(* IEC 61131-3 sources: PLC_ST_Simulator/src/lib/library/standard, 15 files *)

(* ---- FbAxisAbs.st ---- *)
FUNCTION_BLOCK FbAxisAbs
    VAR_INPUT
        iAct : BOOL;
        iAxisNo : INT;
        iSpeed : INT;
        iStop : BOOL;
        iDest : DINT;
    END_VAR
    VAR_OUTPUT
        oBusy : BOOL;
        oDone : BOOL;
        oErr : BOOL;
    END_VAR
    VAR
        done : BOOL;
        (* Mock Logic *)
        tmrDelay : TON;
    END_VAR

    (* Mock Implementation *)
    IF iAct AND NOT oBusy AND NOT oDone THEN
        oBusy := TRUE;
        oErr := FALSE;
    END_IF;

    IF oBusy THEN
        tmrDelay(IN := TRUE, PT := T#500ms);
        IF tmrDelay.Q THEN
            oBusy := FALSE;
            oDone := TRUE;
            tmrDelay(IN := FALSE);
        END_IF;
    ELSE
        tmrDelay(IN := FALSE);
    END_IF;

    IF NOT iAct THEN
        oDone := FALSE;
    END_IF;
END_FUNCTION_BLOCK

(* ---- FbAxisZero.st ---- *)
FUNCTION_BLOCK FbAxisZero
    VAR_INPUT
        iAct : BOOL;
        iAxisNo : INT; (* WORD/Bit String 16 *)
        iHomeSpeed : INT;
        iApproachSpeed : INT;
        iStop : BOOL;
    END_VAR
    VAR_OUTPUT
        oBusy : BOOL;
        oDone : BOOL;
        oErr : BOOL;
    END_VAR
    VAR
        done : BOOL;
        (* Mock Logic *)
        step : INT := 0;
        tmrDelay : TON;
    END_VAR

    (* Mock Implementation *)
    IF iAct AND NOT oBusy AND NOT oDone THEN
        oBusy := TRUE;
        oErr := FALSE;
        step := 1;
    END_IF;

    IF oBusy THEN
        tmrDelay(IN := TRUE, PT := T#1s);
        IF tmrDelay.Q THEN
            oBusy := FALSE;
            oDone := TRUE;
            tmrDelay(IN := FALSE);
        END_IF;
    ELSE
        tmrDelay(IN := FALSE);
    END_IF;

    IF NOT iAct THEN
        oDone := FALSE;
    END_IF;

END_FUNCTION_BLOCK

(* ---- FbCylinder0x1y.st ---- *)
FUNCTION_BLOCK FbCylinder0x1y
    VAR_INPUT
        iAct : BOOL; (* Action Cmd *)
        iOnDelay : INT; (* Sensor On Delay *)
        iOffDelay : INT; (* Sensor Off Delay *)
    END_VAR
    VAR_OUTPUT
        oDevice : BOOL; (* Target Device *)
        oOn : BOOL;
        oOff : BOOL;
    END_VAR
    VAR
        tmrOnDelay : TON;
        tmrOffDelay : TON;
    END_VAR

    oDevice := iAct;

    tmrOnDelay(IN := oDevice, PT := INT_TO_TIME(iOnDelay*10));
    oOn := tmrOnDelay.Q;

    tmrOffDelay(IN := NOT oDevice, PT := INT_TO_TIME(iOffDelay*10));
    oOff := tmrOffDelay.Q;

END_FUNCTION_BLOCK

(* ---- FbCylinder1x1y.st ---- *)
FUNCTION_BLOCK FbCylinder1x1y
    VAR_INPUT
        iAct : BOOL;
        iRst : BOOL;
        iOnDelay : INT;
        iOffDelay : INT;
        iOnTO : INT;
        iOffTO : INT;
        iLimit1 : BOOL;
    END_VAR
    VAR_OUTPUT
        oDevice : BOOL;
        oOn : BOOL;
        oOff : BOOL;
        oErr : BOOL;
        oErrId : INT;
    END_VAR
    VAR
        tmrOn : TON;
        tmrOff : TON;
        tmrOnDelay : TON;
        tmrOffDelay : TON;
    END_VAR

    oDevice := iAct;

    tmrOn(IN := oDevice AND NOT iLimit1, PT:= INT_TO_TIME(iOnTO*10));
    tmrOff(IN := NOT oDevice AND iLimit1, PT:= INT_TO_TIME(iOffTO*10));

    IF iRst AND oErr THEN
        oErr := FALSE;
    END_IF;

    IF tmrOn.Q OR tmrOff.Q THEN
        oErr := TRUE;
    END_IF;

    IF oErr THEN
        IF tmrOff.Q THEN
            oErrId := 20;
        ELSIF tmrOn.Q THEN
            oErrId := 10;
        END_IF;
    ELSE
        oErrId := 0;
    END_IF;

    tmrOnDelay(IN := oDevice AND iLimit1, PT := INT_TO_TIME(iOnDelay*10));
    oOn := tmrOnDelay.Q;

    tmrOffDelay(IN := NOT oDevice, PT := INT_TO_TIME(iOffDelay*10));
    oOff := tmrOffDelay.Q;

END_FUNCTION_BLOCK

(* ---- FbCylinder2x1y.st ---- *)
FUNCTION_BLOCK FbCylinder2x1y
    VAR_INPUT
        iAct : BOOL;
        iRst : BOOL;
        iOnDelay : INT;
        iOffDelay : INT;
        iOnTO : INT;
        iOffTO : INT;
        iLimit1 : BOOL;
        iLimit2 : BOOL;
    END_VAR
    VAR_OUTPUT
        oDevice : BOOL;
        oOn : BOOL;
        oOff : BOOL;
        oErr : BOOL;
        oErrId : INT;
    END_VAR
    VAR
        tmrOn : TON;
        tmrOff : TON;
        tmrErr : TON;
        tmrOnDelay : TON;
        tmrOffDelay : TON;
    END_VAR

    oDevice := iAct;

    tmrOn(IN := oDevice AND NOT iLimit2, PT:= INT_TO_TIME(iOnTO * 10));
    tmrOff(IN := NOT oDevice AND NOT iLimit1, PT := INT_TO_TIME(iOffTO * 10));
    tmrErr(IN := iLimit1 AND iLimit2, PT := T#10s);

    IF iRst AND oErr THEN
        oErr := FALSE;
    END_IF;

    IF tmrOn.Q OR tmrOff.Q OR tmrErr.Q THEN
        oErr := TRUE;
    END_IF;

    IF (oErr) THEN
        IF tmrOn.Q THEN
            oErrId := 10;
        ELSIF  tmrOff.Q THEN
            oErrId := 20;
        END_IF;

        IF tmrErr.Q THEN
            oErrId := 30;
        END_IF;
    ELSE
        oErrId := 0;
    END_IF;

    tmrOnDelay(IN := oDevice AND iLimit2, PT := INT_TO_TIME(iOnDelay*10));
    oOn := tmrOnDelay.Q;

    tmrOffDelay(IN := NOT oDevice AND iLimit1, PT := INT_TO_TIME(iOffDelay*10));
    oOff := tmrOffDelay.Q;

END_FUNCTION_BLOCK

(* ---- FbFeeder.st ---- *)
FUNCTION_BLOCK FbFeeder
    VAR_INPUT
        iAct : BOOL;
        iFull : BOOL;
        iArrived : BOOL;
        iFullOnT : INT;
        iFullOffT : INT;
        iArrivedOnT : INT;
        iSupplyTO : INT;
        iArriveTO : INT;
    END_VAR
    VAR_OUTPUT
        oFeeder : BOOL;
        oLinearFeeder : BOOL;
        oCanPick : BOOL;
        oNeedSupply : BOOL;
        oArriveTO : BOOL;
    END_VAR
    VAR
        tmrArrivedOn : TON;
        tmrFullOn : TON;
        tmrNeedSupply : TON;
        tmrFullOff : TON;
        tmrArriveTO : TON;

        (* Edge helpers *)
        trigFullOff : R_TRIG;
        trigFullOn : R_TRIG;
    END_VAR

    oLinearFeeder := iAct;

    tmrArriveTO(
        IN := iAct AND NOT iArrived,
        PT := INT_TO_TIME(iArriveTO*100));

    tmrArrivedOn(
        IN := iAct AND iArrived,
        PT := INT_TO_TIME(iArrivedOnT*100));

    oCanPick := iAct AND tmrArrivedOn.Q;

    tmrFullOn(
        IN := iAct AND iFull,
        PT := INT_TO_TIME(iFullOnT*100));

    tmrFullOff(
        IN := iAct AND NOT iFull,
        PT := INT_TO_TIME(iFullOffT*100));

    (* Calculate edges *)
    trigFullOff(CLK := tmrFullOff.Q);
    trigFullOn(CLK := tmrFullOn.Q);

    IF iAct THEN
        IF trigFullOff.Q THEN
            oFeeder := TRUE; (* SET *)
        END_IF;

        IF trigFullOn.Q THEN
            oFeeder := FALSE; (* RST *)
        END_IF;
    ELSE
        oFeeder := FALSE; (* RST *)
    END_IF;

    tmrNeedSupply(
        IN := iAct AND oFeeder,
        PT := INT_TO_TIME(iSupplyTO*100));

    oNeedSupply := iAct AND tmrNeedSupply.Q AND (NOT tmrFullOn.Q);

    oArriveTO := tmrArriveTO.Q;

END_FUNCTION_BLOCK

(* ---- FbRotateTable.st ---- *)
FUNCTION_BLOCK FbRotateTable
    VAR_INPUT
        iOrigPos : BOOL;
        iActPos : BOOL;
        iStop : BOOL;
        iRun : BOOL;
        iReset : BOOL;
        iRotateTO : INT;
        iInPosWaitTime : INT;
    END_VAR
    VAR_OUTPUT
        oDevice : BOOL;
        oBusy : BOOL;
        oErr : BOOL;
        oArrived : BOOL;
    END_VAR
    VAR
        rotating : BOOL;
        tmrWaitInPos : TON;
        inPos : BOOL;
        waitInPos : BOOL;
        arrived : BOOL;
        rotate : BOOL;
        reset : BOOL;
        tmrTimeOut : TON;
        tmp : BOOL;

        (* Edge detection helpers *)
        trigRun : R_TRIG;
        trigOrigPos : R_TRIG;
    END_VAR

    (* Pre-calculate edges *)
    trigRun(CLK := iRun);
    rotate := trigRun.Q;
    trigOrigPos(CLK := iOrigPos);

    tmp := (NOT arrived) AND (NOT iStop) AND (rotate OR rotating);
    rotating := tmp;

    (* oDevice output calculation *)
    IF (NOT oErr) AND tmp THEN
        oDevice := TRUE;
    ELSE
        oDevice := FALSE;
    END_IF;

    reset := iReset;
    tmrTimeOut(IN := oDevice AND NOT reset, PT := INT_TO_TIME(iRotateTO * 100)); // Sample says *100? Assuming ms base

    IF NOT reset AND (tmrTimeOut.Q OR oErr) THEN
        oErr := TRUE;
    ELSE
        (* Manual Reset logic might be needed if strictly following Latching logic,
           but here oErr := ... is assignment.
           Sample has oErr := ... (OR oErr), which is self-holding.
           In ST assignment: oErr := ... OR oErr works as hold. *)
         oErr := NOT reset AND (tmrTimeOut.Q OR oErr);
    END_IF;

    inPos := (NOT tmrWaitInPos.Q AND NOT iStop) OR ((rotating AND trigOrigPos.Q) OR inPos);

    waitInPos := (NOT tmrWaitInPos.Q) AND (((NOT iStop) OR ((rotating AND trigOrigPos.Q) OR inPos)) OR waitInPos);

    tmrWaitInPos(IN:= ((inPos AND waitInPos) OR arrived) AND NOT iStop AND NOT tmrWaitInPos.Q, PT := INT_TO_TIME(iInPosWaittime));

    arrived := ((inPos AND waitInPos) OR arrived) AND NOT iStop AND NOT tmrWaitInPos.Q;

    oBusy := rotating AND NOT arrived;

    (* SET/RST translations *)
    IF tmrWaitInPos.Q THEN
        oArrived := TRUE;
    END_IF;

    IF trigRun.Q THEN
        oArrived := FALSE;
    END_IF;

END_FUNCTION_BLOCK

(* ---- FbSysStateProcess.st ---- *)
FUNCTION_BLOCK FbSysStateProcess
    VAR_IN_OUT
        // iStatus : dsSysStatus;
        // iTrig : dsSysTrigger;
    END_VAR

    (* Mock logic *)

END_FUNCTION_BLOCK

(* ---- FbTowerLight.st ---- *)
FUNCTION_BLOCK FbTowerLight
    VAR_INPUT
        // iStatus : dsSysStatus; (* STRUCT not fully supported in simple string parse unless defined *)
        iStopBuzzer : BOOL;
    END_VAR
    VAR_OUTPUT
        // oLights : dsTowerLight;
        hasErr : BOOL;
    END_VAR
    VAR
        keepStopBuzzer : BOOL;
    END_VAR

    (* Mock logic since structs are tricky in this simple setup *)
    hasErr := FALSE;

END_FUNCTION_BLOCK

(* ---- Always.st ---- *)
VAR
    calcA1Speed : BOOL;
    calcA2Speed : BOOL;
    a2HadDone : BOOL;
    axis2ZeroIdx : INT;
    axis1ZeroIdx : INT;
    tmpBool : BOOL;
    st3NextPosIdx : INT;
    manSt5PF : BOOL;
    manSt5LF : BOOL;
    st3StepGoPosIdx : INT;
    idx : INT;
    tmrWaitLetAxis2Down : TON;

    (* Helper vars for edge detection *)
    trigManMode : R_TRIG;
    trigAutoMode : R_TRIG;
    trigSt10Chk : R_TRIG;
    trigFeeder : R_TRIG;
    trigFeederOff : R_TRIG;
    trigRun : R_TRIG;
    trigRotateArrived : R_TRIG;
END_VAR

    tmrSysInit(IN := SM8000, PT:= T#10s);

    sys.EMG := NOT xEmg OR F0;

    IF NOT tmrSysInit.Q THEN
        RETURN;
    END_IF;

    IF sys.EMG THEN
        gSt3NextSide := 0;
        gSt3NeedCheck := TRUE;
    END_IF;

    trigManMode(CLK := sys.ManMode);
    IF trigManMode.Q THEN
        St1PutDone := FALSE;
        St3Done := FALSE;
        St5PutDone := FALSE;
        St6Done := FALSE;
        St7Done := FALSE;
        St8GetDone := FALSE;
        St8NeedGet := FALSE;

        gSt1Seperate := FALSE;
        gSt5Seperate := FALSE;

        St8GetDone := FALSE;
    END_IF;

    (* ALTP(uiLight, yLight); *)
    (* Implementing ALTP (Alternate) logic manually or assuming ALTP FB exists,
       but standard ST doesn't have ALTP. Usage: Toggle yLight on rising edge of uiLight? *)
     (* Assuming uiLight is a button. We need a trigger. *)
     (* For simplicity, skipping ALTP or assuming native support if valid.
        Re-implementing as simple toggle for now: *)
     (* IF trigUiLight.Q THEN yLight := NOT yLight; END_IF; *)

    gAutoCanGoNext := NOT sys.HasError;

    gCanChangePage := gAllStCanCycle;

    tmrSt10Chk(IN:=xSt10Check AND gRotateArrived, PT:=T#0.5s);
    IF gRotateArrived THEN
        IF tmrSt10Chk.Q THEN
            F3 := TRUE;
        END_IF;
    END_IF;

    IF ((uiStartAuto AND (NOT sys.AutoMode)) OR gClearTool) AND
        NOT F3 THEN

        IF NOT sys.HasError AND
            NOT gWaitStopAuto AND gAllStCanCycle AND
            NOT F6 AND
            NOT F7 THEN
            sys.AutoMode := TRUE;
            sys.ManMode := FALSE;
        END_IF;
    END_IF;

    (* SET/RST logic conversion *)
    IF sys.AutoMode AND uiStopAuto AND NOT gWaitStopAuto THEN
        gWaitStopAuto := TRUE;
    END_IF;

    IF sys.AutoMode AND uiStopAuto AND gClearTool THEN
        gClearTool := FALSE;
    END_IF;

    IF uiClearTool AND NOT F3 THEN
        (* CheckHasTool is likely a function call *)
        (* IF CheckHasTool(wDataArray) THEN *)
        (* Assuming CheckHasTool returns BOOL *)
            gClearTool := TRUE;
        (* END_IF; *)
    END_IF;

    gAllStCycleDone :=
        (NOT St1Cycle OR St1PutDone) AND
        (NOT St3Cycle (* OR St3Done*)) AND
        (NOT St5Cycle OR St5PutDone) AND

        ((NOT UseSt6) OR
        (UseSt6 AND NOT St6Cycle)) AND

        NOT St7Cycle AND
        (NOT St8NeedGet OR (St8NeedGet AND St8GetDone)) AND
        NOT St9Cycle;

    gAllStCanCycle :=
        St1InOrg AND
        St3InOrg AND
        St5InOrg AND

        ((NOT UseSt6) OR
        (UseSt6 AND St6InOrg)) AND

        (* St7InOrg AND *)
        St8InOrg AND
        St9InOrg;

    gLight.Yellow :=
        F54 OR
        F55 OR
        F56 OR
        F57;

    gLight.Green :=
        (sys.ManMode AND SM8013) OR
        (sys.AutoMode);

    gLight.Red :=
        SM8013 AND (sys.EMG OR sys.HasError OR sys.HasWarning);

    gBuzzerEnable := NOT uiEnBuzzer;
    gLight.Buzzer := gBuzzerEnable AND
        SM8013 AND (sys.HasWarning OR sys.HasError);

    IF manRotate THEN
        gRotate := TRUE;
        manRotate := FALSE;
    END_IF;

    trigFeeder(CLK := uiFeeder);
    IF trigFeeder.Q THEN
        gSt1RotatoryFeeder := TRUE;
        gSt5RotatoryFeeder := TRUE;

        gSt3Feed := gAllAxisZeroDone AND gA1IO.xReady;
    END_IF;

    trigFeederOff(CLK := uiFeeder); (* This needs falling edge detection *)
    (* Actually LDF is Falling Edge. R_TRIG detects Rising.
       Need F_TRIG for LDF. *)
    (* F_TRIG declaration missing, using logic: *)
    IF (NOT uiFeeder) AND tmpBool(*prev*) THEN
        gSt1RotatoryFeeder := FALSE;
        gSt5RotatoryFeeder := FALSE;
        gSt3Feed := FALSE;

        gSt1Vacuum := FALSE;
        gSt5SquareVacuum := FALSE;
    END_IF;
    tmpBool := uiFeeder; (* Store for falling edge check next cycle *)

    IF gClearDataArray THEN
        FOR idx := 0 TO 9 BY 1 DO
            wDataArray[idx] := 0;
        END_FOR;
        gClearDataArray := FALSE;
    END_IF;

    RotateTable(
        iOrigPos:= xIndexOrg,
        iActPos:= xIndexAct,
        iRun:= gRotate AND (NOT sys.Error),
        iRotateTO:= wRotateTO,
        iInPosWaitTime:= wRotateOnPosWaitT,
        iReset := ResetAlarm,
        oDevice => yIndex);

    IF RotateTable.oBusy THEN
        gRotate := FALSE;
    END_IF;

    trigRotateArrived(CLK := RotateTable.oArrived);
    IF trigRotateArrived.Q THEN
        gRotateArrived := TRUE;
    END_IF;

    (* Cylinders *)
    cySt1Down(
        iAct := gSt1Down,
        iRst := ResetAlarm,
        iLimit1 := xSt1DownOrg,
        iLimit2 := xSt1DownAct,
        oDevice =>ySt1Down,
        iOnTO := wSt1DownTO,
        iOffTO := wSt1DownTO,
        iOnDelay := wSt1DownOnT,
        iOffDelay := wSt1DownOffT);

    cySt1Forward(
        iAct := gSt1Forward,
        iRst := ResetAlarm,
        iLimit1 := xSt1ForwardOrg,
        iLimit2 := xSt1ForwardAct,
        oDevice =>ySt1Forward,
        iOnTO := wSt1ForwardTO,
        iOffTO := wSt1ForwardTO,
        iOnDelay := wSt1ForwardOnT,
        iOffDelay := wSt1ForwardOffT);

    cySt1Clamp(
        iAct := gSt1Clamp,
        oDevice =>ySt1Clamp,
        iOnDelay := wSt1ClampOnT,
        iOffDelay := wSt1ClampOffT);

    cySt1ClampRotate(
        iAct := gSt1ClampRotate,
        iRst := ResetAlarm,
        iLimit1 := xSt1ClampRotateOrg,
        iLimit2 := xSt1ClampRotateAct,
        oDevice =>ySt1ClampRotate,
        iOnTO := wSt1ClampRotateTO,
        iOffTO := wSt1ClampRotateTO,
        iOnDelay := wSt1ClampRotateOnT,
        iOffDelay := wSt1ClampRotateOffT);

    cySt1Seperate(
        iAct := gSt1Seperate,
        iRst := ResetAlarm,
        iLimit1 := xSt1SeperateOrg,
        iLimit2 := xSt1SeperateAct,
        oDevice =>ySt1Seperate,
        iOnTO := wSt1SeperateTO,
        iOffTO := wSt1SeperateTO,
        iOnDelay := wSt1SeperateOnT,
        iOffDelay := wSt1SeperateOffT);

    cySt3Down(
        iAct := gSt3Down,
        iRst := ResetAlarm,
        iLimit1 := xSt3DownOrg,
        iLimit2 := xSt3DownAct,
        oDevice =>ySt3Down,
        iOnTO := wSt3DownTO,
        iOffTO := wSt3DownTO,
        iOnDelay := wSt3DownOnT,
        iOffDelay := wSt3DownOffT);

    cySt3Forward(
        iAct := gSt3Forward,
        iRst := ResetAlarm,
        iLimit1 := xSt3ForwardOrg,
        iLimit2 := xSt3ForwardAct,
        oDevice =>ySt3Forward,
        iOnTO := wSt3ForwardTO,
        iOffTO := wSt3ForwardTO,
        iOnDelay := wSt3ForwardOnT,
        iOffDelay := wSt3ForwardOffT);

    cySt3Suck(
        iAct := gSt3Suck,
        iRst := ResetAlarm,
        iLimit1 := xSt3SuckOrg,
        oDevice => ySt3Suck,
        iOnDelay := wSt3SuckOnT,
        iOffDelay := wSt3SuckOffT,
        iOnTO := wSt3SuckTO,
        iOffTO := wSt3SuckTO);

    cySt5Suck(
        iAct := gSt5Suck,
        iRst := ResetAlarm,
        iLimit1 := xSt5SuckOrg,
        oDevice => ySt5Vacuum,
        iOnDelay := wSt5SuckOnT,
        iOffDelay := wSt5SuckOffT,
        iOnTO := wSt5SuckTO,
        iOffTO := wSt5SuckTO);

    cySt5Down(
        iAct := gSt5Down,
        iRst := ResetAlarm,
        iLimit1 := xSt5DownOrg,
        iLimit2 := xSt5DownAct,
        oDevice =>ySt5Down,
        iOnTO := wSt5DownTO,
        iOffTO := wSt5DownTO,
        iOnDelay := wSt5DownOnT,
        iOffDelay := wSt5DownOffT);

    cySt5Forward(
        iAct := gSt5Forward,
        iRst := ResetAlarm,
        iLimit1 := xSt5ForwardOrg,
        iLimit2 := xSt5ForwardAct,
        oDevice =>ySt5Forward,
        iOnTO := wSt5ForwardTO,
        iOffTO := wSt5ForwardTO,
        iOnDelay := wSt5ForwardOnT,
        iOffDelay := wSt5ForwardOffT);

    cySt5Seperate(
        iAct := gSt5Seperate,
        iRst := ResetAlarm,
        iLimit1 := xSt5SeperateOrg,
        iLimit2 := xSt5SeperateAct,
        oDevice =>ySt5Seperate,
        iOnTO := wSt5SeperateTO,
        iOffTO := wSt5SeperateTO,
        iOnDelay := wSt5SeperateOnT,
        iOffDelay := wSt5SeperateOffT);

    cySt6Down(
        iAct := gSt6Down,
        iRst := ResetAlarm,
        iLimit1 := xSt6DownOrg,
        iLimit2 := xSt6DownAct,
        oDevice =>ySt6Down,
        iOnTO := wSt6DownTO,
        iOffTO := wSt6DownTO,
        iOnDelay := wSt6DownOnT,
        iOffDelay := wSt6DownOffT);

    cySt8Down(
        iAct := gSt8Down,
        iRst := ResetAlarm,
        iLimit1 := xSt8DownOrg,
        iLimit2 := xSt8DownAct,
        oDevice =>ySt8Down,
        iOnTO := wSt8DownTO,
        iOffTO := wSt8DownTO,
        iOnDelay := wSt8DownOnT,
        iOffDelay := wSt8DownOffT);

    cySt8Forward(
        iAct := gSt8Forward,
        iRst := ResetAlarm,
        iLimit1 := xSt8ForwardOrg,
        iLimit2 := xSt8ForwardAct,
        oDevice =>ySt8Forward,
        iOnTO := wSt8ForwardTO,
        iOffTO := wSt8ForwardTO,
        iOnDelay := wSt8ForwardOnT,
        iOffDelay := wSt8ForwardOffT);

    cySt8Clamp(
        iAct := gSt8Clamp,
        oDevice =>ySt8Clamp,
        iOnDelay := wSt8ClampOnT,
        iOffDelay := wSt8ClampOffT);

    cySt9Up(
        iAct := gSt9Up,
        iRst := ResetAlarm,
        iLimit1 := xSt9UpOrg,
        iLimit2 := xSt9UpAct,
        oDevice =>ySt9Up,
        iOnTO := wSt9UpTO,
        iOffTO := wSt9UpTO,
        iOnDelay := wSt9UpOnT,
        iOffDelay := wSt9UpOffT);

    cySt9BlowAir(
        iAct := gSt9BlowAir,
        oDevice =>ySt9BlowAir,
        iOnDelay := wSt9BlowAirOnT,
        iOffDelay := wSt9BlowAirOffT);

    rfSt1(
        iAct:= gSt1RotatoryFeeder AND NOT ResetAlarm,
        iFull:= xSt1LF_Full,
        iArrived:= xSt1LF_FeedIn,
        iFullOnT:= wSt1FullOnT,
        iFullOffT:= wSt1FullOffT,
        iArrivedOnT:= wSt1FeedInOnT,
        oCanPick => gSt1CanPick,
        oFeeder => gSt1PF,
        oLinearFeeder => gSt1LF,
        iSupplyTO:= wSt1FullTO,
        iArriveTO:= wSt1FeedInTO);

    trigSt1CanPick(CLK := gSt1CanPick);
    IF trigSt1CanPick.Q THEN
        gSt1Vacuum := TRUE;
    END_IF;

    ySt1PF := gSt1PF OR (manSt1PF AND sys.ManMode);
    ySt1LF := gSt1LF OR (manSt1LF AND sys.ManMode);

    rfSt5(
        iAct:= gSt5RotatoryFeeder AND NOT ResetAlarm,
        iFull:= xSt5LF_Full,
        iArrived:= xSt5LF_FeedIn,
        iFullOnT:= wSt5FullOnT,
        iFullOffT:= wSt5FullOffT,
        iArrivedOnT:= wSt5FeedInOnT,
        oCanPick => gSt5CanPick,
        oFeeder => gSt5PF,
        oLinearFeeder => gSt5LF,
        iSupplyTO:= wSt5FullTO,
        iArriveTO:= wSt5FeedInTO);

    ySt5PF := gSt5PF OR (manSt5PF AND sys.ManMode);
    ySt5LF := gSt5LF OR (manSt5LF AND sys.ManMode);

    ySt1Vacuum := gSt1Vacuum;
    ySt5VacuumBreak := gSt5VacuumBreak;

    ySt5SquareVacuum := gSt5SquareVacuum;

(* ---- Auto.st ---- *)
VAR
    autoGoNext : BOOL;
    idx : INT;
    trigAutoMode : R_TRIG;
    trigSM8012 : R_TRIG;
END_VAR

    IF NOT tmrSysInit.Q THEN
        RETURN;
    END_IF;

    IF NOT xBackDoor AND NOT ResetAlarm THEN
        errDoorOpen := TRUE;
    END_IF;

    trigAutoMode(CLK := sys.AutoMode);
    IF trigAutoMode.Q THEN
        wAutoIdx := 10;
        uiFeeder := TRUE;
    END_IF;

    IF NOT sys.AutoMode THEN
        RETURN;
    END_IF;

    trigSM8012(CLK := SM8012);
    IF NOT errDoorOpen THEN
        IF gCalcCycleTime AND trigSM8012.Q THEN
            wCycleTime := wCycleTime + 1;
        END_IF;
    END_IF;

    CASE wAutoIdx OF
    10:
        (* rotate plate *)
        gRotate := TRUE;
        gRotateArrived := FALSE;

        autoGoNext := TRUE;
    20:
        IF RotateTable.oBusy THEN
            gRotate := FALSE;

            (* shift data *)
            FOR idx := 1 TO 9 BY 1 DO
                wDataArray[10-idx] := wDataArray[9-idx];
            END_FOR;

            wDataArray[0] := 0;

            autoGoNext := TRUE;
        ELSIF RotateTable.oErr THEN
            wAutoIdx := NG_STEP;
        END_IF;
    30:
        (* index table rotating, check which station should act. *)
        (* station 1 *)
        IF NOT gClearTool THEN
            wDataArray[0] := 10;
            autoSt1Cycle := NOT gClearTool;
        END_IF;

        (* station 3 *)
        IF (wDataArray[2] = (20+ STEP_OK)) THEN
            autoSt3Cycle := TRUE;
        END_IF;

        (* station 5 *)
        IF wDataArray[4] = (40+STEP_OK) THEN
             autoSt5Cycle := TRUE;
        END_IF;

        autoGoNext := TRUE;
    40:
        (* index table arrived, check which station should act. *)
        IF gRotateArrived  THEN
            (* station 6 *)
            IF wDataArray[5] = (50+STEP_OK) THEN
                IF UseSt6 THEN
                    autoSt6Cycle := TRUE;
                ELSE
                    wDataArray[5] := 60+STEP_OK;
                END_IF;
            END_IF;

            (* station 8 - ok *)
            IF wDataArray[7] = (70+STEP_OK) OR St7ResultOK THEN
                St7ResultOK := FALSE;

                St8GetDone := FALSE;
                St8NeedGet := TRUE;
            ELSE
                St8NeedGet := FALSE;
            END_IF;

            (* station 9 - ng *)
            IF (wDataArray[8] >= TOOL_NG) THEN
                autoSt9Cycle := TRUE;
            END_IF;

            autoGoNext := TRUE;
        END_IF;
    50:
        IF gAllStCycleDone THEN

            IF St1PutDone THEN
                wDataArray[0] := 10+STEP_OK;
            END_IF;

            (* IF gSt2HasTool THEN *)
            IF xSt2Check THEN
                wDataArray[1] := 20+STEP_OK;
            END_IF;

            IF St3Done THEN
                IF gSt3CurIsBackSide THEN
                    wDataArray[2] := 903;
                    wSt3CountNG := wSt3CountNG + 1;
                ELSE
                    wDataArray[2] := 30+STEP_OK;
                    wSt3CountNG := 0;
                END_IF;

                IF wSt3CountNG >= CONTINUS_NG_TARGET THEN
                    St3ContNG := TRUE;
                ELSE
                    St3ContNG := FALSE;
                END_IF;

                gSt3CurIsBackSide := FALSE;
            END_IF;

            (* station 4 *)
            IF (wDataArray[3] = (30+STEP_OK)) THEN
                (* IF gSt4HasTool THEN *)
                IF xSt4Check THEN
                    wDataArray[3] := 40+STEP_OK;
                    wSt4CountNG := 0;
                ELSE
                    wDataArray[3] := 904;
                    wSt4CountNG := wSt4CountNG + 1;
                END_IF;

                IF wSt4CountNG >= CONTINUS_NG_TARGET THEN
                    St4ContNG := TRUE;
                ELSE
                    St4ContNG := FALSE;
                END_IF;
            END_IF;

            IF St5PutDone THEN
                wDataArray[4] := 50+STEP_OK;
            END_IF;

            IF St6Done THEN
                wDataArray[5] := 60+STEP_OK;
            END_IF;

            (* station 7 *)
            IF (wDataArray[6] = (60+STEP_OK)) THEN
                IF st7HasTool AND st7ToolOk THEN
                    St7ResultOK := TRUE;
                ELSE
                    St7ResultOK := FALSE;
                END_IF;

                IF St7ResultOK THEN
                    wDataArray[6] := 70+STEP_OK;
                    wSt7CountNG := 0;
                ELSE
                    wDataArray[6] := 907;
                    wSt7CountNG := wSt7CountNG + 1;
                END_IF;

                IF wSt7CountNG >= CONTINUS_NG_TARGET THEN
                    St7ContNG := TRUE;
                ELSE
                    St7ContNG := FALSE;
                END_IF;
            END_IF;

            IF St8GetDone THEN
                wDataArray[7] := 0;
                wProductOkCount := wProductOkCount + 1;
                wTotalOkCnt := wTotalOkCnt + 1;
            END_IF;

            IF St9Done THEN
                wDataArray[8] := 0;
                wProductNgCount := wProductNgCount + 1;
            END_IF;

            St1PutDone := FALSE;
            St3Done := FALSE;
            St5PutDone := FALSE;
            St6Done := FALSE;
            St7Done := FALSE;
            St8GetDone := FALSE;
            St9Done := FALSE;
            St8NeedGet := FALSE;

            IF gEnStopCount THEN
                IF wProductOkCount >= wStopMachineNumber THEN
                    gTargetCounted := TRUE;
                    gWaitStopAuto := TRUE;
                END_IF;
            END_IF;

            IF gClearTool THEN
                IF CheckHasTool(wDataArray) = FALSE THEN
                    gClearTool := FALSE;
                    gWaitStopAuto := TRUE;
                END_IF;
            END_IF;

            wAutoIdx := 60;
        END_IF;	(* all cycle done *)
    60:
        (* non resident and non target counted *)
        IF (NOT F3) AND
            (NOT F4) AND
            NOT St3ContNG AND
            NOT St4ContNG AND
            NOT St7ContNG THEN

            IF NOT gWaitStopAuto THEN
                wAutoIdx := 10;
            ELSE
                wAutoIdx := OK_STEP;
            END_IF;
        END_IF;
    END_CASE;

    IF St8NeedGet AND (NOT St8GetDone) AND gRotateArrived AND (NOT St8Cycle) THEN
        autoSt8Cycle := TRUE;
    END_IF;

    IF wAutoIdx = OK_STEP THEN
        wAutoIdx := 0;
        sys.AutoMode := FALSE;
        sys.ManMode := TRUE;
        gWaitStopAuto := FALSE;
        uiFeeder := FALSE;

        gClearTool := FALSE;

    ELSIF wAutoIdx = NG_STEP THEN
        IF gAutoCanGoNext THEN
            wAutoIdx := 0;
        END_IF;
    END_IF;

    IF autoGoNext THEN
        IF gAutoCanGoNext THEN
            wAutoIdx := wAutoIdx + 10;
            autoGoNext := FALSE;
        END_IF;
    END_IF;

(* ---- Error.st ---- *)
    IF NOT tmrSysInit.Q THEN
        RETURN;
    END_IF;

    ResetAlarm := uiResetAlarm;
    (* BKRSTP(ResetAlarm, 100, F0); *)
    (* Replaced BKRSTP with TODO or explicit reset if crucial *)
    IF ResetAlarm THEN
       (* Mock clearing F0..100 *)
       F0 := FALSE;
       F1 := FALSE;
       (* ... *)
    END_IF;

    sys.HasError :=
        F0 OR
        F1 OR
        (* F2 *)
        errDoorOpen OR
        (* F3 OR *)
        F4 OR
        F5 OR
        F6 OR
        F7
        ;

    sys.HasWarning := SM8048;

    IF sys.EMG THEN
        sys.AutoMode := FALSE;
        sys.ManMode := TRUE;
        gWaitStopAuto := FALSE;
        gClearTool := FALSE;

        gSt1RotatoryFeeder := FALSE;
        gSt5RotatoryFeeder := FALSE;
        gSt3Feed := FALSE;

        gSt1Vacuum := FALSE;
        uiFeeder := FALSE;

        St1Cycle := FALSE;
        St3Cycle := FALSE;
        St5Cycle := FALSE;
        St6Cycle := FALSE;
        St7Cycle := FALSE;
        St8Cycle := FALSE;
        St9Cycle := FALSE;

        gAllAxisZeroDone := FALSE;
    END_IF;

    IF ResetAlarm THEN
        IF St2ContNG THEN
            wSt2CountNG := 0;
        END_IF;

        IF St3ContNG THEN
            wSt3CountNG := 0;
        END_IF;

        IF St4ContNG THEN
            wSt4CountNG := 0;
        END_IF;

        IF St7ContNG THEN
            wSt7CountNG := 0;
        END_IF;

        St3ContNG := FALSE;
        St4ContNG := FALSE;
        St7ContNG := FALSE;
    ELSE
        IF F58 THEN St3ContNG := TRUE; END_IF;
        IF F59 THEN St4ContNG := TRUE; END_IF;
        IF F63 THEN St7ContNG := TRUE; END_IF;

        IF F0 THEN sys.EMG := TRUE; END_IF;
        IF F1 THEN RotateTable.oErr := TRUE; END_IF;

        IF gEnStopCount AND gTargetCounted THEN
            F4 := TRUE;
            gTargetCounted := FALSE;
        END_IF;

        IF NOT X26 THEN F5 := TRUE; END_IF;
        IF NOT gA1ZeroDone THEN F6 := TRUE; END_IF;
        IF NOT gA2ZeroDone THEN F7 := TRUE; END_IF;

        IF cySt1Down.oErr THEN
            IF cySt1Down.oErrId = ErrCyOn THEN F10 := TRUE; END_IF;
            IF cySt1Down.oErrId = ErrCyOff THEN F11 := TRUE; END_IF;
            IF cySt1Down.oErrId = ErrCyBoth THEN F12 := TRUE; END_IF;
        END_IF;

        (* ... more Cylinder error mapping ... *)
    END_IF;

(* ---- Init.st ---- *)
    yLight := TRUE;
    sys.ManMode := TRUE;
    (* gCanChangePage := TRUE; *)

    ySt3ServoServoBrake := TRUE;
    ySt3ServoServoOn := TRUE;

    IF dwSt3Seperation = 0 THEN
        dwSt3Seperation := 4;
    END_IF;

    SM8049 := TRUE;

(* ---- Manual.st ---- *)
    IF (NOT tmrSysInit.Q) OR sys.EMG OR (NOT sys.ManMode) THEN
        RETURN;
    END_IF;

    (* DMOV substitutions - assuming standard assignments work for now *)
    wProductOkCount := 0;
    wProductNgCount := 0;
    wTotalOkCnt := 0;

    IF uiResetAllSt THEN
        uiSt1Reset := TRUE;
        uiSt3Reset := TRUE;
        uiSt5Reset := TRUE;
        uiSt6Reset := TRUE;
        uiSt7Reset := TRUE;
        uiSt8Reset := TRUE;
        uiSt9Reset := TRUE;
    END_IF;

    CASE wPageIndex OF
    11:
        IF NOT St1Cycle THEN
            (* ALTP replacement with IFs if needed, or assume ALTP is supported/mocked *)
            (* ALTP in Manual usually means button toggle. *)
            (* ALTP(M50 AND cySt1Seperate.oOn, gSt1Down); *)
        END_IF;
        uiSt1Reset := uiStReset;
    13:
        IF NOT St3Cycle THEN
            (* Mock ALTPs *)
        END_IF;

    END_CASE;

    (* can change page *)
    M81 :=
        (wPageIndex=11 AND St1Cycle) OR
        (wPageIndex=13 AND St3Cycle) OR
        SM8001;

    IF uiSt1Reset THEN
        gSt1Down := FALSE;
        gSt1Forward := FALSE;
        gSt1Clamp := FALSE;
        gSt1ClampRotate := FALSE;
        gSt1Seperate := FALSE;

        St1Cycle := FALSE;

        manSt1PF := FALSE;
        manSt1LF := FALSE;
        gSt1PF := FALSE;
        gSt1LF := FALSE;
        gSt1Vacuum := FALSE;

        uiSt1Reset := FALSE;
    END_IF;

    IF uiSt3Reset THEN
        gSt3Down := FALSE;
        gSt3Forward := FALSE;
        gSt3Suck := FALSE;
        gSt3GoSafeHeight := FALSE;

        St3Cycle := FALSE;

        gSt3Feed := FALSE;
        uiSt3Reset := FALSE;
    END_IF;

(* ---- St1.st ---- *)
VAR
    canGoNext : BOOL;
    goNext : BOOL;
    goNg : BOOL;
END_VAR

    (* Station 1 Logic *)
    IF St1Cycle THEN

        IF wSt1Index = OK_STEP THEN
            St1Cycle := FALSE;
            wSt1Index := 0;

        ELSIF wSt1Index = NG_STEP THEN
            IF canGoNext THEN
                wSt1Index := wSt1LastIndex;
                wSt1LastIndex := 0;
            END_IF;
        END_IF;

        IF sys.AutoMode THEN
            IF gSt1CanPick AND NOT gSt1Seperate THEN
                gSt1Seperate := TRUE;
            END_IF;
        END_IF;

        CASE wSt1Index OF
        10:
            IF sys.AutoMode THEN
                wDataArray[0] := 10 + STEP_BUSY;
            END_IF;
            IF NOT F54 THEN
                IF gSt1CanPick OR sys.ManMode THEN
                    gSt1Seperate := TRUE;
                END_IF;
            END_IF;

            IF cySt1Seperate.oOn THEN
                goNext := TRUE;
            ELSIF cySt1Seperate.oErr THEN
                gSt1Seperate := FALSE;
                goNg := TRUE;
            END_IF;
        20:
            gSt1Down := TRUE;

            IF cySt1Down.oOn THEN
                goNext := TRUE;
            ELSIF cySt1Down.oErr THEN
                gSt1Down := FALSE;
                goNg := TRUE;
            END_IF;
        30:
            gSt1Clamp := TRUE;
            IF cySt1Clamp.oOn THEN
                gSt1Vacuum := FALSE;
                goNext := TRUE;
            END_IF;
        40:	(* up *)
            gSt1Down := FALSE;
            IF cySt1Down.oOff THEN
                gSt1Seperate := FALSE;
                goNext := TRUE;
            ELSIF cySt1Down.oErr THEN
                goNg := TRUE;
            END_IF;
        50:	(* rotate, forward *)
            gSt1ClampRotate := TRUE;
            gSt1Forward := TRUE;
            IF cySt1ClampRotate.oOn THEN
                goNext := TRUE;
            ELSIF cySt1ClampRotate.oErr THEN
                gSt1Forward := FALSE;
                goNg := TRUE;
            END_IF;
        60:	(* forward *)
            goNext := TRUE;
            gSt1Forward := TRUE;

            IF cySt1Forward.oOn THEN
                goNext := TRUE;
            ELSIF cySt1Forward.oErr THEN
                gSt1Forward := FALSE;
                goNg := TRUE;
            END_IF;

        70:	(* down *)
            IF sys.ManMode THEN
                gSt1Down := TRUE;
            ELSIF sys.AutoMode THEN
                IF gRotateArrived THEN gSt1Down := TRUE; END_IF;
            END_IF;

            IF cySt1Down.oOn THEN
                goNext := TRUE;
            ELSIF cySt1Down.oErr THEN
                gSt1Down := FALSE;
                goNg := TRUE;
            END_IF;
        80:	(* clamp off *)
            gSt1Clamp := FALSE;
            IF cySt1Clamp.oOff THEN goNext := TRUE; END_IF;

        90:	(* up *)
            gSt1Down := FALSE;
            IF cySt1Down.oOff THEN
                St1PutDone := TRUE;
                goNext := TRUE;
            ELSIF cySt1Down.oErr THEN
                goNg := TRUE;
            END_IF;
        100: (* back *)
            gSt1Forward := FALSE;
            gSt1ClampRotate := FALSE;

            IF cySt1Forward.oOff AND cySt1ClampRotate.oOff THEN
                goNext := TRUE;
            ELSIF cySt1Forward.oErr THEN
                goNg := TRUE;
            END_IF;
        110:
            wSt1Index := OK_STEP;
        END_CASE;

        IF goNg THEN
            wSt1LastIndex := wSt1Index;
            wSt1Index := NG_STEP;
            goNg := FALSE;
        END_IF;

        IF goNext AND canGoNext THEN
            wSt1Index := wSt1Index + 10;
            goNext := FALSE;
        END_IF;
    END_IF;

    St1InOrg :=
        cySt1Down.oOff AND
        cySt1Forward.oOff AND
        cySt1Clamp.oOff AND
        cySt1ClampRotate.oOff AND
        SM8000;

    canGoNext :=
        NOT sys.HasError AND
        NOT cySt1Down.oErr AND
        NOT cySt1Forward.oErr AND
        NOT cySt1ClampRotate.oErr AND
        NOT cySt1Seperate.oErr AND
        SM8000;
